// TIA Portal V20 export
FUNCTION_BLOCK "LConSMC_MovAverage"   // FB32043, SCL
// stored: Access Published, IsIECCheckEnabled true, MemoryReserve 100, SetENOAutomatically true
   VAR_INPUT
      enable { ExternalAccessible := 'False'; ExternalVisible := 'False'; ExternalWritable := 'False'} : Bool := TRUE;
      updateConfig { ExternalAccessible := 'False'; ExternalVisible := 'False'; ExternalWritable := 'False'} : Bool;
      sampleMode { ExternalAccessible := 'False'; ExternalVisible := 'False'; ExternalWritable := 'False'} : UInt;
      inputSignal { ExternalAccessible := 'False'; ExternalVisible := 'False'; ExternalWritable := 'False'} : LReal;
      subsetLength { ExternalAccessible := 'False'; ExternalVisible := 'False'; ExternalWritable := 'False'} : UInt;
      samplingFactor { ExternalAccessible := 'False'; ExternalVisible := 'False'; ExternalWritable := 'False'} : UInt;
      setTimePeriod { ExternalAccessible := 'False'; ExternalVisible := 'False'; ExternalWritable := 'False'} : Time;
      cycleTime { ExternalAccessible := 'False'; ExternalVisible := 'False'; ExternalWritable := 'False'} : UDInt;   // Cycle time in ns
   END_VAR
   VAR_OUTPUT
      error { ExternalAccessible := 'False'; ExternalVisible := 'False'; ExternalWritable := 'False'} : Bool;
      errorID { ExternalAccessible := 'False'; ExternalVisible := 'False'; ExternalWritable := 'False'} : DWord := 16#0000_0000;
      samplingTime { ExternalAccessible := 'False'; ExternalVisible := 'False'; ExternalWritable := 'False'} : LReal := 1.0;
      timePeriod { ExternalAccessible := 'False'; ExternalVisible := 'False'; ExternalWritable := 'False'} : LReal := 10.0;
      shiftedInputSignal { ExternalAccessible := 'False'; ExternalVisible := 'False'; ExternalWritable := 'False'} : LReal;
      movingAverage { ExternalAccessible := 'False'; ExternalVisible := 'False'; ExternalWritable := 'False'} : LReal;
   END_VAR
   VAR
      statUpdateConfigOld { ExternalAccessible := 'False'; ExternalVisible := 'False'; ExternalWritable := 'False'} : Bool;
      statEnableOld { ExternalAccessible := 'False'; ExternalVisible := 'False'; ExternalWritable := 'False'} : Bool;
      statError { ExternalAccessible := 'False'; ExternalVisible := 'False'; ExternalWritable := 'False'} : Bool;
      statSum { ExternalAccessible := 'False'; ExternalVisible := 'False'; ExternalWritable := 'False'} : LReal;
      statSignalBufferSum { ExternalAccessible := 'False'; ExternalVisible := 'False'; ExternalWritable := 'False'} : Array[1.."LCON_STATEVAL_MAX_BUFFERLENGTH"] of LReal;
      statSamplingFactor { ExternalAccessible := 'False'; ExternalVisible := 'False'; ExternalWritable := 'False'} : UInt;
      statSubsetLength { ExternalAccessible := 'False'; ExternalVisible := 'False'; ExternalWritable := 'False'} : UInt;
      instfbUpdateConfig { ExternalAccessible := 'False'; ExternalVisible := 'False'; ExternalWritable := 'False'} : "LConSMC_UpdateConfigOfStatisticCalc";
      instfbSumCalc { ExternalAccessible := 'False'; ExternalVisible := 'False'; ExternalWritable := 'False'} : "LConSMC_SumCalc";
      statEnableRisingEdge { ExternalAccessible := 'False'; ExternalVisible := 'False'; ExternalWritable := 'False'} : Bool;
      statCurrentSubLen { ExternalAccessible := 'False'; ExternalVisible := 'False'; ExternalWritable := 'False'} : UInt;
   END_VAR
   VAR CONSTANT
      FB_ID : DWord := 16#0426_0000;
      INIT_TIMEPERIOD : Time := T#10MS;
      INIT_MULT_OF_SAMPLINGRATE : UInt := 1;
   END_VAR
BEGIN
   //===========================================================================================================
   // SIEMENS AG
   // (c)Copyright 2019  All Rights Reserved
   //-----------------------------------------------------------------------------------------------------------
   //  file name:      LDrvOpt_MovAverage (Motion Control Application Cycle)
   //  library:        LDrvOpt
   //  system:         SIMATIC TIA PORTAL V15
   //  version:        V1.0.0   
   //  restrictions:   Must be called in PreIpo
   //  requirements:   /
   //  functionality:  This function block calculates the moving average for any input signal by an user defined 
   //                  subset n. It also delivers the centered input signal for the moving average.
   //                  Any changes of the subset length during calculation causes no peak. It may be used to smooth
   //                  loop control signals.    
   //        
   //                  The implemented algorithm calculates as shown in the following formula:            
   //                  µ_(n)     =     (1 / n) * SUM[i = k-n...k] x_i
   //------------------------------------------------------------------------------------------------------------
   //  change log table:
   //  version     date            experts in charge           changes applied
   //  01.00.00    15.03.19        APC Erlangen                create
   //============================================================================================================

   //----------------------------------------------------------------------
   //RESET SETTINGS AND ERRORS AFTER RISING EDGE OF ENABLE
   //----------------------------------------------------------------------
   IF (#enable AND NOT #statEnableOld) THEN
       // start calculation in default mode after Reset und clear errors
       #statEnableOld := #enable;
       #statEnableRisingEdge := TRUE;
   ELSE
       #statEnableRisingEdge := FALSE;
   END_IF;

   IF (NOT #enable) THEN
       #statEnableOld := #enable;

       //Reset outputs
       #statError := FALSE;
       #error := FALSE;
       #errorID := 16#0000_0000;
       #samplingTime := 0.0;
       #timePeriod := 0.0;
       #shiftedInputSignal := 0.0;
       #movingAverage := 0.0;
   END_IF;

   //----------------------------------------------------------------------
   //UPDATE CONFIGURATION FOR AVERAGING
   //----------------------------------------------------------------------
   // Detect rising edge of UpdateConfig
   IF ((#updateConfig AND NOT #statUpdateConfigOld) OR #statEnableRisingEdge) THEN

       #instfbUpdateConfig(
                           fb_ID := #FB_ID,
                           cascadeCalculation := FALSE,
                           sampleMode := #sampleMode,
                           maxBufferLengthMain := "LCON_STATEVAL_MAX_BUFFERLENGTH",
                           inSubsetLengthMain := #subsetLength,
                           setTimePeriod := #setTimePeriod,
                           inSamplingFactor := #samplingFactor,
                           cycleTime := #cycleTime,
                           error => #statError,
                           errorID => #errorID,
                           outSamplingFactorMain => #statSamplingFactor,
                           outSubsetLengthMain => #statSubsetLength,
                           samplingTime => #samplingTime,
                           timePeriod => #timePeriod
       );

       #statUpdateConfigOld := #updateConfig;

   END_IF;

   IF (NOT #updateConfig) THEN
       #statUpdateConfigOld := #updateConfig;
   END_IF;

   //----------------------------------------------------------------------
   //DETERMINE MOVING AVERAGE
   //----------------------------------------------------------------------
   // If an error is queued the calculation will be stopped to prevent CPU stopp
   IF (NOT #statError AND #enable) THEN

       // Calculate Average (a wrong configuration doesn't stopp the calculation)
       #instfbSumCalc(
                      enable := #enable,
                      inputSignal := #inputSignal,
                      inSubsetLength := #statSubsetLength,
                      inRateOfSumCalc := #statSamplingFactor,
                      signalBuffer := #statSignalBufferSum,
                      sum => #statSum,
                      shiftedInputSignal => #shiftedInputSignal,
                      outSubsetLength => #statCurrentSubLen
       );

       // Calculate moving average of sum
       #movingAverage := (1.0 / #statCurrentSubLen) * #statSum;

       // determine the current time periode of the subset
       //#timePeriod := #samplingTime * #statCurrentSubLen;    //actual time period during init
   END_IF;
   #error := #statError;
END_FUNCTION_BLOCK
